FUNCTION_BLOCK Hall
VAR_INPUT
END_VAR
VAR_OUTPUT
END_VAR
VAR
	keypad01 : Keypad;
	lamp01:	DigitalLight;
	lamp02:	DigitalLight;
	lamp03:	DigitalLight;
	dimmer01 : Dimmer;
	
END_VAR


	EL1008_01;
	EL1008_02;
	EL1008_03;
	EL2008_01;
	EL2008_02;
	EL4004_01;
	
	lamp01(input:=	EL1008_01[0], keyType:= );
	EL2008_01[0]	:=	lamp01.output;
	EL2008_01[1]	:=	lamp01.output;
	
	lamp02(input:=	EL1008_01[1], keyType:= );
	EL2008_01[2]	:=	lamp02.output;
	
	lamp03(input:=	EL1008_01[2], keyType:= );
	EL2008_01[3]	:=	lamp03.output;
	
	dimmer01(input01:= EL1008_02[0], input02:= EL1008_02[1]);
	EL4004_01[0]	:= dimmer01.output;

END_FUNCTION_BLOCK

(* stored: Version 1.1.0.1, ProductVersion 3.1.4024.13
   POU Hall: Id {4b00a001-43ea-4b70-b88a-a8dcac3d88f3}, SpecialFunc None *)
